// Mitsubishi GX Works2 project: 28-06-2LAB3   PLC: FX3G

PROGRAM MAIN
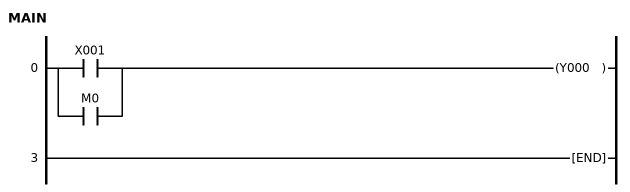
0     LD      X001
      OR      M0
      OUT     Y000
3     END
END_PROGRAM
